(* CODESYS project CtaAppStufenManagement_1.0.0.2.library
   Description: Stufenmanagement Library der CTA
   Version: 1.0.0.2
   Title: CtaAppStufenManagement
   Author: SIS
   DocFormat: reStructuredText
   LanguageModelAttribute: qualified-access-only
   Placeholder: CtaAppStufenManagement
   DefaultNamespace: CtaAppStufenManagement
   CompiledLibraryCompatibilityVersion: CODESYS V3.5 SP16 Patch 3
   Company: CTA

Project tree, tasks and I/O mapping:
  libraries: Standard, 3.5.18.0 (System); CtaSysConfig, 1.0.0.2 (CTA); CtaSysTypes, 1.0.0.0 (CTA); CtaVisSymbols, 1.0.0.0 (CTA); CtaVisApps, 1.0.0.0 (CTA); CtaVisHelp, 1.0.0.0 (CTA); CtaVisUser, 1.0.0.0 (CTA); VisuSymbols, 4.5.0.0 (System)
  40 Visualizations/
    visualisation VIS_Manager_rEck
    Dialog/
      visualisation DIA_MANAGER
    visualisation VIS_Manager
  00000000-0000-0000-0000-000000000000|D:\CoDeSys\LibrariesV3\trunk\Intern\CAA\CAA Template\3.4.0.0 draft\Placeholder.xml
  00000000-0000-0000-0000-000000000000|D:\CoDeSys\LibrariesV3\trunk\Intern\CAA\CAA Template\3.2.0.3 draft\Prefix.pdf
  00000000-0000-0000-0000-000000000000|D:\CoDeSys\LibrariesV3\trunk\Intern\CAA\CAA Template\3.5.2.0 draft\Placeholder.xml
  20 Structs/
    data type TYPE_OF_ENGINE_MANAGEMENT
    data type scParameter
  50 Images/
  10 Documenation/
    global variables VersionHistory
    global variables readMe
  21 Interface/
    Group/
      GroupBase/
        interface ITF_GROUPBASE: IS_NOT_RELEVANT_TO_CHECK, SET_OPERATION_MODES, proiAcknowledge, prorAcknowledge, proxAcknowledge, IS_NOT_RELEVANT_TO_RELEASE, proiAvaiable, prorAvaiable, proxAvaiable, proxLockDown, IS_NOT_RELEVANT_TO_ACKNOWLEDGE
      GroupLeader/
        Circuit/
          interface ITF_CIRCUIT: GET_ANZ_AVAIABLE, GET_ANZ_ACKNOWLEDGE, GET_ANZ_RELEASE, CIRCUIT_NR, ALL_OFF, IS_RELEVANT_TO_RELEASE, GET_ENGINE_STATE, RELEASE_ENGINE, LOWERBOUND, UPPERBOUND, metSetRelease, proxRelease, GET_ANZ_LOCKDOWN, SET_HZ_SCALE, SET_ENGINE_STATE, prorRelease, proxAcknowledge
      GroupMember/
        Hydraulics/
          interface ITF_HYDRA: MEMBER_OF, IS_ADDED_TO_NESSESARY, CALCULATET_TIME_TILL_RUN, ESTIMATET_TIME_TILL_RUN, metSetRelease, proxRelease
    Manager/
      interface ITF_MANAGER: ADD_CLIENT
  11 Library Parameter/
  12 Konstanten/
    global variables GVL_CONSTANT
  60 Textlisten/
    text list TypeOfEngineManagement
  13 Globale Variablen/
  text list GlobalTextList
  5ce3da45-db07-42e7-a21c-a00fff4ed8f6|C:\Users\sis\Downloads\dip-switch.svg
  5ce3da45-db07-42e7-a21c-a00fff4ed8f6|C:\Users\sis\Downloads\lightning-bolt-circle.svg
  30 Program Organization Units/
    Group/
      GroupBase/
        function block GROUPBASE [ST]: IS_NOT_RELEVANT_TO_CHECK, SET_OPERATION_MODES, IS_NOT_RELEVANT_TO_RELEASE, proenRelease, proenCheck, proiAcknowledge, prorAcknowledge, proxAcknowledge, proiAvaiable, prorAvaiable, proxAvaiable, proxLockDown, IS_NOT_RELEVANT_TO_ACKNOWLEDGE
      GroupLeader/
        Help/
          function block ENGINE [ST]: GET_ANZ_AVAIABLE, GET_ANZ_ACKNOWLEDGE, GET_ANZ_RELEASE, GET_ANZ_LOCKDOWN, SET_ENGINE_STATE, GET_ENGINE_STATE, RELEASE_ENGINE, LOWERBOUND, UPPERBOUND, SET_HZ_SCALE
        Circuit/
          function block CIRCUIT [ST]: IS_RELEVANT_TO_RELEASE, proiAvaiable, SET_ENGINE_STATE, prorRelease, metSetRelease, proxRelease, GET_ANZ_AVAIABLE, GET_ANZ_ACKNOWLEDGE, GET_ANZ_RELEASE, CIRCUIT_NR, ALL_OFF, GET_ENGINE_STATE, RELEASE_ENGINE, LOWERBOUND, UPPERBOUND, GET_ANZ_LOCKDOWN, SET_HZ_SCALE, proxAvaiable, proxAcknowledge, proiAcknowledge
      GroupMember/
        Help/
          function block GROUPMEMBER [ST]
          function block TIME_TIL_RUN [ST]: CALCULATET_TIME_TILL_RUN, ESTIMATET_TIME_TILL_RUN
        Hydraulics/
          function block HYDRA [ST]: IS_ADDED_TO_NESSESARY, MEMBER_OF, FB_INIT, CALCULATET_TIME_TILL_RUN, ESTIMATET_TIME_TILL_RUN, metSetRelease, proxRelease
    Manager/
      function block MANAGER [ST]: GET_NEXT_ENGINE_TO_RUN, GET_NEXT_ENGINE_TO_OFF, MANAGEMENT, CHECK_RELEASE_CHANGE, UPDATE_AT_THE_END, ACKNOWLEDGE, RELEASE, LOCKDOWN, AVAIABLE, ADD_CLIENT, actParameter
  5ce3da45-db07-42e7-a21c-a00fff4ed8f6|C:\Users\sis\Downloads\sine-wave.svg
  5ce3da45-db07-42e7-a21c-a00fff4ed8f6|C:\Users\sis\Downloads\eye.svg
  5ce3da45-db07-42e7-a21c-a00fff4ed8f6|C:\Users\sis\Downloads\lan.svg
*)

// 20 Structs/TYPE_OF_ENGINE_MANAGEMENT
{attribute 'qualified_only'}
TYPE TYPE_OF_ENGINE_MANAGEMENT :
(
	RUN_1BY1 	:= 0,
	RUN_EQUAL	:= 1
);
END_TYPE

// 20 Structs/scParameter
TYPE scParameter :
	STRUCT
		fbtZuschaltSperrzeit		:	CtaSysConfig.fbTIME;
		fbiTypeOfEngineManagement	:	CtaSysConfig.fbINT;
	END_STRUCT
END_TYPE

// 10 Documenation/VersionHistory
(* 

.. image:: ../../Images/CTA_Logo.jpg
   :align: right
   :width: 15% 

**Vorlage**   


============ =========== =========== ============================================
**Date**     **Version** **Author**  **Change**
------------ ----------- ----------- --------------------------------------------
04.03.2021   0.0.0.0     SIS         Vorlage erstellt

============ =========== =========== ============================================


*)
VAR_GLOBAL
    stInfo : STRING:= '0.0.0.0, Vorlage, CTA';
END_VAR

// 10 Documenation/readMe
(*

**ReadMe**
 
|	**Empfehlung**
|
|	Die Bibliothek CtaAppStufenManagement dient dem Management der ganzen Maschine, sie Schaltet beispielsweise Kreise und Stufen frei.
|	Instanzieren Sie den CtaAppStufenManagement.MANAGER in ihrem Funktionsbaustein oder POU beispielsweise als Manager
|	Deklarieren Sie die Struktur Variable welche als Parameter und zur ansteuerung dienen wie im Code beispiel.
|  
| *Beispiel* 

+-----------------------+---------------------------------------------------------------------------------------------------------------------------------------------------------------------------------------------------------------------------------------------------------------------------------------------------------------------------------------------------------------------------------------------------------------------------------------+
| Beschreibung          |  Code                                                                                                                                                                                                                                                                                                                                                                                                                                 |
+=======================+=======================================================================================================================================================================================================================================================================================================================================================================================================================================+
| Pou oder SmFb         | .. code-block:: codesys                                                                                                                                                                                                                                                                                                                                                                                                               |
|                       |                                                                                                                                                                                                                                                                                                                                                                                                                                       |
|                       |	// Deklaration als VAR im POU oder dem selbsterstellten Funktionsbaustein                                                                                                                                                                                                                                                                                                                                                       	|
|                       |   VAR   																																																																																																								|
|						|	    (*Maschinen Management*)																																																		 																																																|
|						|		MANAGER			: CtaAppStufenManagement.MANAGER;                                                                                                                                                                                                                                                                                                                                                             				 	|
|						|																																																																																																										|
+-----------------------+---------------------------------------------------------------------------------------------------------------------------------------------------------------------------------------------------------------------------------------------------------------------------------------------------------------------------------------------------------------------------------------------------------------------------------------+
| Code für Init         | .. code-block:: codesys                                                                                                                                                                                                                                                                                                                                                                                                               |
|                       |   																																																																																																									|
| 						|	// Kopieren des nachfolgenden Codes in eine Action zur Initialisierung der Parameter. Zum Beispiel actConfig.																																																																														|
|                       |	{region "Maschinen Management"}                                                                                                                                                                                                                                                                                                                                                                                                     |
|						|		MANAGER.scParameter.fbtZuschaltSperrzeit               		(_wertInit :=	 T#5m														);		//P1 Zeit die vergeht bis die nächste Stufe zugeschalten werden kann																																																			|
|						|		MANAGER.scParameter.fbiTypeOfEngineManagement				(_wertInit :=	 	0		, _minInit :=			, _maxInit :=			);		//P2 0 = Ausschöpfung des Kreises / 1 = Beliebig nach verfügbarkeit																																																				| 
|						|	{endregion}                                                                                                                                                      																																																																	| 
+-----------------------+---------------------------------------------------------------------------------------------------------------------------------------------------------------------------------------------------------------------------------------------------------------------------------------------------------------------------------------------------------------------------------------------------------------------------------------+
*)                                                                                                                                                                                                                                                                                                                                                                                                                                                               
 VAR_GLOBAL                                                                                                                                                                                                                                                                                                                                                                                                                                                      
    xReadMeDone              :   BOOL;                                                                                                                                                                                                                                                                                                                                                                                                                           
END_VAR

// 12 Konstanten/GVL_CONSTANT
{attribute 'qualified_only'}
VAR_GLOBAL CONSTANT
	MAX_GROUPS	:	USINT	:= 4;
	MAX_ENGINE	:	USINT	:= 4;
END_VAR

// 21 Interface/Group/GroupBase/ITF_GROUPBASE
INTERFACE ITF_GROUPBASE EXTENDS __SYSTEM.IQueryInterface

PROPERTY IS_NOT_RELEVANT_TO_CHECK : BOOL
GET
END_GET
SET
END_SET
END_PROPERTY

METHOD SET_OPERATION_MODES
VAR_INPUT
	enCheckIn		:	INT;
	enReleaseIn		:	INT;
END_VAR
END_METHOD

{attribute 'monitoring' := 'call'}
PROPERTY proiAcknowledge : INT
SET
END_SET
GET
END_GET
END_PROPERTY

PROPERTY prorAcknowledge : REAL
SET
END_SET
GET
END_GET
END_PROPERTY

{attribute 'monitoring' := 'call'}
PROPERTY proxAcknowledge : BOOL
SET
END_SET
GET
END_GET
END_PROPERTY

PROPERTY IS_NOT_RELEVANT_TO_RELEASE : BOOL
GET
END_GET
SET
END_SET
END_PROPERTY

{attribute 'monitoring' := 'call'}
PROPERTY proiAvaiable : INT
SET
END_SET
GET
END_GET
END_PROPERTY

PROPERTY prorAvaiable : REAL
SET
END_SET
GET
END_GET
END_PROPERTY

{attribute 'monitoring' := 'call'}
PROPERTY proxAvaiable : BOOL
SET
END_SET
GET
END_GET
END_PROPERTY

{attribute 'monitoring' := 'call'}
PROPERTY proxLockDown : BOOL
SET
END_SET
GET
END_GET
END_PROPERTY

PROPERTY IS_NOT_RELEVANT_TO_ACKNOWLEDGE : BOOL
SET
END_SET
GET
END_GET
END_PROPERTY

END_INTERFACE

// 21 Interface/Manager/ITF_MANAGER
INTERFACE ITF_MANAGER EXTENDS __SYSTEM.IQueryInterface

METHOD ADD_CLIENT : BOOL
VAR_INPUT
	ITF_GROUP_BASE_IN	:	ITF_GROUPBASE;
END_VAR
END_METHOD

END_INTERFACE

// 21 Interface/Group/GroupLeader/Circuit/ITF_CIRCUIT
INTERFACE ITF_CIRCUIT EXTENDS ITF_GROUPBASE

PROPERTY GET_ANZ_AVAIABLE : UINT
GET
END_GET
END_PROPERTY

PROPERTY GET_ANZ_ACKNOWLEDGE : UINT
GET
END_GET
END_PROPERTY

PROPERTY GET_ANZ_RELEASE : UINT
GET
END_GET
END_PROPERTY

PROPERTY CIRCUIT_NR : USINT
GET
END_GET
END_PROPERTY

METHOD ALL_OFF : BOOL
VAR_INPUT
END_VAR
END_METHOD

PROPERTY IS_RELEVANT_TO_RELEASE : BOOL
GET
END_GET
SET
END_SET
END_PROPERTY

METHOD GET_ENGINE_STATE : BOOL
VAR_INPUT
	usiNr				:	USINT;
END_VAR
VAR_OUTPUT	    	
	xAvaiable			:	BOOL;
	xRelease			:	BOOL;
	rRelease			:	REAL;
	xAcknowledge		:	BOOL;
	rAcknowledge		:	REAL;
	xLockDown			:	BOOL;
	udiRunTime			:	UDINT;
	udiRunTimeTillOn	:	UDINT;
END_VAR
END_METHOD

METHOD RELEASE_ENGINE
VAR_INPUT
	usiNr		:	USINT;
	xRelease	:	BOOL;
END_VAR
END_METHOD

PROPERTY LOWERBOUND : DINT
GET
END_GET
END_PROPERTY

PROPERTY UPPERBOUND : DINT
GET
END_GET
END_PROPERTY

METHOD metSetRelease
VAR_INPUT
	xReleaseCircuit	:	BOOL;	
END_VAR
END_METHOD

{attribute 'monitoring' := 'call'}
PROPERTY proxRelease : BOOL
GET
END_GET
END_PROPERTY

PROPERTY GET_ANZ_LOCKDOWN : UINT
GET
END_GET
END_PROPERTY

METHOD SET_HZ_SCALE
VAR_INPUT
	scHz		:	CtaSysTypes.scHzParameter;
END_VAR
END_METHOD

METHOD SET_ENGINE_STATE 
VAR_INPUT
	usiNr		:	USINT;
	xAvaiable	:	BOOL;
	xAcknowledge:	BOOL;
	rAcknowledge:	REAL;
	xLockDown	:	BOOL;
	rNewRelease	:	REAL;
END_VAR
VAR_OUTPUT
	xRelease	:	BOOL;
	rRelease	:	REAL;
	scHz		:	CtaSysTypes.scHzParameter;
END_VAR
END_METHOD

PROPERTY prorRelease : REAL
SET
END_SET
GET
END_GET
END_PROPERTY

{attribute 'monitoring' := 'call'}
PROPERTY proxAcknowledge : BOOL
SET
END_SET
GET
END_GET
END_PROPERTY

END_INTERFACE

// 21 Interface/Group/GroupMember/Hydraulics/ITF_HYDRA
INTERFACE ITF_HYDRA EXTENDS ITF_GROUPBASE

METHOD MEMBER_OF : BOOL
VAR_INPUT
	usiGROUP_NR	:	USINT;
END_VAR
END_METHOD

PROPERTY IS_ADDED_TO_NESSESARY : BOOL
SET
END_SET
GET
END_GET
END_PROPERTY

PROPERTY CALCULATET_TIME_TILL_RUN : TIME
SET
END_SET
GET
END_GET
END_PROPERTY

PROPERTY ESTIMATET_TIME_TILL_RUN : TIME
SET
END_SET
GET
END_GET
END_PROPERTY

METHOD metSetRelease
VAR_INPUT
	usiNr		:	USINT;
	xRelease	:	BOOL;	
END_VAR
END_METHOD

{attribute 'monitoring' := 'call'}
PROPERTY proxRelease : BOOL
GET
END_GET
END_PROPERTY

END_INTERFACE

// 30 Program Organization Units/Group/GroupBase/GROUPBASE
FUNCTION_BLOCK GROUPBASE IMPLEMENTS ITF_GROUPBASE
VAR_INPUT
	ITF_MANAGER_IN			:	ITF_MANAGER;
END_VAR    
VAR_OUTPUT
	xAvaiable					:	BOOL;
	iAvaiable					:	INT;
	rAvaiable					:	REAL;
	xAcknowledge				:	BOOL;
	iAcknowledge				:	INT;
	rAcknowledge				:	REAL;
	xLockDown					:	BOOL;
END_VAR         		         		
VAR                 		
	enCheck						:	INT;
	enRelease					:	INT;	
	xIsNotRelevantToRelease		:	BOOL;
	xIsNotRelevantToCheck		:	BOOL;
	xIsNotRelevantToAcknowledge :	BOOL;
END_VAR

IF __QUERYINTERFACE(ITF_MANAGER_IN,ITF_MANAGER_IN) THEN
	ITF_MANAGER_IN.ADD_CLIENT(THIS^);	
END_IF;

PROPERTY IS_NOT_RELEVANT_TO_CHECK : BOOL
GET
IS_NOT_RELEVANT_TO_CHECK := xIsNotRelevantToCheck;
END_GET
SET
xIsNotRelevantToCheck := IS_NOT_RELEVANT_TO_CHECK;
END_SET
END_PROPERTY

METHOD SET_OPERATION_MODES
VAR_INPUT
	enCheckIn		:	INT;
	enReleaseIn		:	INT;
END_VAR
enCheck 	:= enCheckIn;
enRelease 	:= enReleaseIn;
END_METHOD

PROPERTY IS_NOT_RELEVANT_TO_RELEASE : BOOL
GET
IS_NOT_RELEVANT_TO_RELEASE := xIsNotRelevantToRelease;
END_GET
SET
xIsNotRelevantToRelease := IS_NOT_RELEVANT_TO_RELEASE;
END_SET
END_PROPERTY

{attribute 'monitoring' := 'call'}
PROPERTY proenRelease : INT
GET
proenRelease := enRelease;
END_GET
END_PROPERTY

{attribute 'monitoring' := 'call'}
PROPERTY proenCheck : INT
GET
proenCheck := enCheck;
END_GET
END_PROPERTY

{attribute 'monitoring' := 'call'}
PROPERTY proiAcknowledge : INT
SET
iAcknowledge := proiAcknowledge;
END_SET
GET
proiAcknowledge := iAcknowledge;
END_GET
END_PROPERTY

PROPERTY prorAcknowledge : REAL
SET
rAcknowledge := prorAcknowledge;
END_SET
GET
prorAcknowledge := rAcknowledge;
END_GET
END_PROPERTY

{attribute 'monitoring' := 'call'}
PROPERTY proxAcknowledge : BOOL
SET
xAcknowledge := proxAcknowledge;
END_SET
GET
proxAcknowledge := xAcknowledge;
END_GET
END_PROPERTY

{attribute 'monitoring' := 'call'}
PROPERTY proiAvaiable : INT
SET
iAvaiable := proiAvaiable;
END_SET
GET
proiAvaiable := iAvaiable;
END_GET
END_PROPERTY

PROPERTY prorAvaiable : REAL
SET
rAvaiable := prorAvaiable;
END_SET
GET
prorAvaiable := rAvaiable;
END_GET
END_PROPERTY

{attribute 'monitoring' := 'call'}
PROPERTY proxAvaiable : BOOL
SET
xAvaiable := proxAvaiable;
END_SET
GET
proxAvaiable := xAvaiable;
END_GET
END_PROPERTY

{attribute 'monitoring' := 'call'}
PROPERTY proxLockDown : BOOL
SET
xLockDown := proxLockDown;
END_SET
GET
proxLockDown := xLockDown;
END_GET
END_PROPERTY

PROPERTY IS_NOT_RELEVANT_TO_ACKNOWLEDGE : BOOL
GET
IS_NOT_RELEVANT_TO_ACKNOWLEDGE := xIsNotRelevantToAcknowledge;
END_GET
SET
xIsNotRelevantToAcknowledge := IS_NOT_RELEVANT_TO_ACKNOWLEDGE;
END_SET
END_PROPERTY

END_FUNCTION_BLOCK

// 30 Program Organization Units/Group/GroupLeader/Circuit/CIRCUIT
FUNCTION_BLOCK CIRCUIT EXTENDS GROUPBASE IMPLEMENTS ITF_CIRCUIT
VAR_INPUT
	usiNr	:	USINT;
END_VAR
VAR_OUTPUT
END_VAR
VAR
	xRelease				:	BOOL;
	rRelease				:	REAL;
	xIsRelevantToRelease	:	BOOL;
	ENGINE					:	ENGINE;
	diFor					:	DINT;
END_VAR

SUPER^();

PROPERTY IS_RELEVANT_TO_RELEASE : BOOL
SET
xIsRelevantToRelease := IS_RELEVANT_TO_RELEASE;
END_SET
GET
IS_RELEVANT_TO_RELEASE := xIsRelevantToRelease;
END_GET
END_PROPERTY

{attribute 'monitoring' := 'call'}
PROPERTY proiAvaiable : INT
SET
iAvaiable := proiAvaiable;
END_SET
GET
iAvaiable	:= TO_INT(GET_ANZ_AVAIABLE);
proiAvaiable := iAvaiable;
END_GET
END_PROPERTY

METHOD SET_ENGINE_STATE 
VAR_INPUT
	usiNr		:	USINT;
	xAvaiable	:	BOOL;
	xAcknowledge:	BOOL;
	rAcknowledge:	REAL;
	xLockDown	:	BOOL;
	rNewRelease	:	REAL;
END_VAR
VAR_OUTPUT
	xRelease	:	BOOL;
	rRelease	:	REAL;
	scHz		:	CtaSysTypes.scHzParameter;
END_VAR
ENGINE.SET_ENGINE_STATE(usiNr 			:= usiNr,
						xAvaiable 		:= xAvaiable,
						xAcknowledge	:= xAcknowledge,
						rAcknowledge	:= rAcknowledge,
						xLockDown		:= xLockDown,
						rNewRelease		:= rNewRelease,
						xRelease		=> xRelease,
						rRelease		=> rRelease,
						scHz			=> scHz);
END_METHOD

PROPERTY prorRelease : REAL
SET
rRelease := prorRelease;
END_SET
GET
prorRelease := rRelease;
END_GET
END_PROPERTY

METHOD metSetRelease
VAR_INPUT
	xReleaseCircuit	:	BOOL;	
END_VAR
xRelease := xReleaseCircuit;
IF NOT xRelease THEN
	ALL_OFF();
END_IF;
END_METHOD

{attribute 'monitoring' := 'call'}
PROPERTY proxRelease : BOOL
GET
proxRelease := xRelease;
END_GET
END_PROPERTY

PROPERTY GET_ANZ_AVAIABLE : UINT
GET
VAR
	diForTemp	:	DINT;
END_VAR
GET_ANZ_AVAIABLE := ENGINE.GET_ANZ_AVAIABLE;
END_GET
END_PROPERTY

PROPERTY GET_ANZ_ACKNOWLEDGE : UINT
GET
VAR
	diForTemp	:	DINT;
END_VAR
GET_ANZ_ACKNOWLEDGE := ENGINE.GET_ANZ_ACKNOWLEDGE;
END_GET
END_PROPERTY

PROPERTY GET_ANZ_RELEASE : UINT
GET
VAR
	diForTemp	:	DINT;
END_VAR
GET_ANZ_RELEASE := ENGINE.GET_ANZ_RELEASE;
END_GET
END_PROPERTY

PROPERTY CIRCUIT_NR : USINT
GET
CIRCUIT_NR := usiNr;
END_GET
END_PROPERTY

METHOD ALL_OFF : BOOL
VAR_INPUT
END_VAR
VAR
	diLowerBound	:	DINT;
	diUpperBound	:	DINT;
	diForTemp1		:	DINT;
END_VAR
(* Stopp ALL *)
FOR diForTemp1 := ENGINE.LOWERBOUND TO ENGINE.UPPERBOUND DO
	ENGINE.RELEASE_ENGINE(TO_USINT(diForTemp1),FALSE);
END_FOR;
END_METHOD

METHOD GET_ENGINE_STATE : BOOL
VAR_INPUT
	usiNr		:	USINT;
END_VAR
VAR_OUTPUT	    	
	xAvaiable			:	BOOL;
	xRelease			:	BOOL;
	rRelease			:	REAL;
	xAcknowledge		:	BOOL;
	rAcknowledge		:	REAL;
	xLockDown			:	BOOL;
	udiRunTime			:	UDINT;
	udiRunTimeTillOn	:	UDINT;
END_VAR
ENGINE.GET_ENGINE_STATE(usiNr 				:= usiNr,
						xAvaiable			=> xAvaiable,
						xRelease			=> xRelease,
						rRelease			=> rRelease,
						xAcknowledge		=> xAcknowledge,
						rAcknowledge		=> rAcknowledge,
						xLockDown			=> xLockDown,
						udiRunTime			=> udiRunTime,
						udiRunTimeTillOn	=> udiRunTimeTillOn);
END_METHOD

METHOD RELEASE_ENGINE
VAR_INPUT
	usiNr		:	USINT;
	xRelease	:	BOOL;
END_VAR
ENGINE.RELEASE_ENGINE(	usiNr		:= usiNr,
						xRelease 	:= xRelease);
END_METHOD

PROPERTY LOWERBOUND : DINT
GET
LOWERBOUND := ENGINE.LOWERBOUND;
END_GET
END_PROPERTY

PROPERTY UPPERBOUND : DINT
GET
UPPERBOUND := ENGINE.UPPERBOUND;
END_GET
END_PROPERTY

PROPERTY GET_ANZ_LOCKDOWN : UINT
GET
GET_ANZ_LOCKDOWN := ENGINE.GET_ANZ_LOCKDOWN;
END_GET
END_PROPERTY

METHOD SET_HZ_SCALE
VAR_INPUT
	scHz		:	CtaSysTypes.scHzParameter;
END_VAR
ENGINE.SET_HZ_SCALE(scHz);
END_METHOD

{attribute 'monitoring' := 'call'}
PROPERTY proxAvaiable : BOOL
SET
xAvaiable := proxAvaiable;
END_SET
GET
proxAvaiable := SUPER^.proxAvaiable;
END_GET
END_PROPERTY

{attribute 'monitoring' := 'call'}
PROPERTY proxAcknowledge : BOOL
SET
xAcknowledge := proxAcknowledge;
END_SET
GET
proxAcknowledge := xAcknowledge;
END_GET
END_PROPERTY

{attribute 'monitoring' := 'call'}
PROPERTY proiAcknowledge : INT
SET
iAcknowledge := proiAcknowledge;
END_SET
GET
iAcknowledge := TO_INT(GET_ANZ_ACKNOWLEDGE);
proiAcknowledge := iAcknowledge;
END_GET
END_PROPERTY

END_FUNCTION_BLOCK

// 30 Program Organization Units/Group/GroupLeader/Help/ENGINE
FUNCTION_BLOCK ENGINE
VAR_INPUT
END_VAR
VAR_OUTPUT
END_VAR
VAR
	scHzAll				:	CtaSysTypes.scHzParameter;
	AY_XRELEASE			:	ARRAY[1..GVL_CONSTANT.MAX_ENGINE] OF BOOL;
	AY_RRELEASE			:	ARRAY[1..GVL_CONSTANT.MAX_ENGINE] OF REAL;
	AY_XAVAIABLE		:	ARRAY[1..GVL_CONSTANT.MAX_ENGINE] OF BOOL;
	AY_XACKNOWLEDGE		:	ARRAY[1..GVL_CONSTANT.MAX_ENGINE] OF BOOL;
	AY_XACKNOWLEDGEOLD	:	ARRAY[1..GVL_CONSTANT.MAX_ENGINE] OF BOOL;
	AY_RACKNOWLEDGE		:	ARRAY[1..GVL_CONSTANT.MAX_ENGINE] OF REAL;
	AY_LOCKDOWN			:	ARRAY[1..GVL_CONSTANT.MAX_ENGINE] OF BOOL;
	AY_RUN_TIME			:	ARRAY[1..GVL_CONSTANT.MAX_ENGINE] OF UDINT;
	AY_RUN_TIME_TILL_ON	:	ARRAY[1..GVL_CONSTANT.MAX_ENGINE] OF UDINT;
	AY_TON_RUN_TIME		:	ARRAY[1..GVL_CONSTANT.MAX_ENGINE] OF Standard.TON;
END_VAR

PROPERTY GET_ANZ_AVAIABLE : UINT
GET
VAR
	diForTemp	:	DINT;
END_VAR
GET_ANZ_AVAIABLE := 0;
FOR diForTemp := LOWER_BOUND(AY_XAVAIABLE,1) TO UPPER_BOUND(AY_XAVAIABLE,1) DO
	IF AY_XAVAIABLE[diForTemp] THEN
		GET_ANZ_AVAIABLE := GET_ANZ_AVAIABLE + 1;
	END_IF;
END_FOR;
END_GET
END_PROPERTY

PROPERTY GET_ANZ_ACKNOWLEDGE : UINT
GET
VAR
	diForTemp	:	DINT;
END_VAR
GET_ANZ_ACKNOWLEDGE := 0;
FOR diForTemp := LOWER_BOUND(AY_XACKNOWLEDGE,1) TO UPPER_BOUND(AY_XACKNOWLEDGE,1) DO
	IF AY_XACKNOWLEDGE[diForTemp] THEN
		GET_ANZ_ACKNOWLEDGE := GET_ANZ_ACKNOWLEDGE + 1;
	END_IF;
END_FOR;
END_GET
END_PROPERTY

PROPERTY GET_ANZ_RELEASE : UINT
GET
VAR
	diForTemp	:	DINT;
END_VAR
GET_ANZ_RELEASE := 0;
FOR diForTemp := LOWER_BOUND(AY_XRELEASE,1) TO UPPER_BOUND(AY_XRELEASE,1) DO
	IF AY_XRELEASE[diForTemp] THEN
		GET_ANZ_RELEASE := GET_ANZ_RELEASE + 1;
	END_IF;
END_FOR;
END_GET
END_PROPERTY

PROPERTY GET_ANZ_LOCKDOWN : UINT
GET
VAR
	diForTemp	:	DINT;
END_VAR
GET_ANZ_LOCKDOWN := 0;
FOR diForTemp := LOWER_BOUND(AY_LOCKDOWN,1) TO UPPER_BOUND(AY_LOCKDOWN,1) DO
	IF AY_LOCKDOWN[diForTemp] THEN
		GET_ANZ_LOCKDOWN := GET_ANZ_LOCKDOWN + 1;
	END_IF;
END_FOR;
END_GET
END_PROPERTY

METHOD SET_ENGINE_STATE 
VAR_INPUT
	usiNr		:	USINT;
	xAvaiable	:	BOOL;
	xAcknowledge:	BOOL;
	rAcknowledge:	REAL;
	xLockDown	:	BOOL;
	rNewRelease	:	REAL;
END_VAR
VAR_OUTPUT
	xRelease	:	BOOL;
	rRelease	:	REAL;
	scHz		:	CtaSysTypes.scHzParameter;
END_VAR
(* Avaiable *)
IF usiNr >= LOWER_BOUND(AY_XAVAIABLE,1) AND usiNr <= UPPER_BOUND(AY_XAVAIABLE,1) THEN
	AY_XAVAIABLE[usiNr] := xAvaiable;
END_IF;

(* Acknowledge *)
IF usiNr >= LOWER_BOUND(AY_XACKNOWLEDGE,1) AND usiNr <= UPPER_BOUND(AY_XACKNOWLEDGE,1) THEN
	AY_XACKNOWLEDGEOLD[usiNr] 	:= AY_XACKNOWLEDGE[usiNr];
	AY_XACKNOWLEDGE[usiNr] 		:= xAcknowledge;
END_IF;
IF usiNr >= LOWER_BOUND(AY_RACKNOWLEDGE,1) AND usiNr <= UPPER_BOUND(AY_RACKNOWLEDGE,1) THEN
	AY_RACKNOWLEDGE[usiNr] := rAcknowledge;
END_IF

(* LockDown *)
IF usiNr >= LOWER_BOUND(AY_LOCKDOWN,1) AND usiNr <= UPPER_BOUND(AY_LOCKDOWN,1) THEN
	AY_LOCKDOWN[usiNr] := xLockDown;
	IF xLockDown THEN
		AY_XRELEASE[usiNr] := FALSE;
	END_IF;
END_IF;

(* Release *)
IF usiNr >= LOWER_BOUND(AY_XRELEASE,1) AND usiNr <= UPPER_BOUND(AY_XRELEASE,1) THEN
	(* No release if no more acknowledge *)
	IF AY_XRELEASE[usiNr] AND AY_XRELEASE[usiNr] = AY_XACKNOWLEDGEOLD[usiNr] AND NOT AY_XACKNOWLEDGE[usiNr] THEN
		AY_XRELEASE[usiNr] := FALSE;
	END_IF;	
	xRelease := AY_XRELEASE[usiNr] AND NOT xLockDown;
ELSE
	xRelease := FALSE;
END_IF;
IF usiNr >= LOWER_BOUND(AY_RRELEASE,1) AND usiNr <= UPPER_BOUND(AY_RRELEASE,1) THEN
	AY_RRELEASE[usiNr]	:= rNewRelease;
	rRelease 			:= AY_RRELEASE[usiNr];
ELSE
	rRelease := 0;
END_IF;

(* TIME *)
IF usiNr >= LOWER_BOUND(AY_RUN_TIME,1) AND usiNr <= UPPER_BOUND(AY_RUN_TIME,1) THEN
	AY_TON_RUN_TIME[usiNr](IN := NOT AY_TON_RUN_TIME[usiNr].Q AND xRelease AND xAcknowledge,
						   PT := T#1M);
	IF AY_TON_RUN_TIME[usiNr].Q THEN
		AY_RUN_TIME[usiNr] 			:= AY_RUN_TIME[usiNr] + 1;
		AY_RUN_TIME_TILL_ON[usiNr] 	:= AY_RUN_TIME_TILL_ON[usiNr] + 1;
	END_IF;
	IF NOT xRelease THEN
		AY_RUN_TIME_TILL_ON[usiNr] 	:= 0;
	END_IF;
END_IF;

scHz := scHzAll;
END_METHOD

METHOD GET_ENGINE_STATE : BOOL
VAR_INPUT
	usiNr			:	USINT;
END_VAR         	
VAR_OUTPUT	    	
	xAvaiable			:	BOOL;
	xRelease			:	BOOL;
	rRelease			:	REAL;
	xAcknowledge		:	BOOL;
	rAcknowledge		:	REAL;
	xLockDown			:	BOOL;
	udiRunTime			:	UDINT;
	udiRunTimeTillOn	:	UDINT;
END_VAR
(* Avaiable *)
IF usiNr >= LOWER_BOUND(AY_XAVAIABLE,1) AND usiNr <= UPPER_BOUND(AY_XAVAIABLE,1) THEN
	xAvaiable := AY_XAVAIABLE[usiNr];
END_IF;

(* Release *)
IF usiNr >= LOWER_BOUND(AY_XRELEASE,1) AND usiNr <= UPPER_BOUND(AY_XRELEASE,1) THEN
	xRelease := AY_XRELEASE[usiNr];
END_IF;

(* Release *)
IF usiNr >= LOWER_BOUND(AY_RRELEASE,1) AND usiNr <= UPPER_BOUND(AY_RRELEASE,1) THEN
	rRelease := AY_RRELEASE[usiNr];
END_IF;

(* Acknowledge *)
IF usiNr >= LOWER_BOUND(AY_XACKNOWLEDGE,1) AND usiNr <= UPPER_BOUND(AY_XACKNOWLEDGE,1) THEN
	xAcknowledge := AY_XACKNOWLEDGE[usiNr];
END_IF;
IF usiNr >= LOWER_BOUND(AY_RACKNOWLEDGE,1) AND usiNr <= UPPER_BOUND(AY_RACKNOWLEDGE,1) THEN
	rAcknowledge := AY_RACKNOWLEDGE[usiNr];
END_IF

(* LockDown *)
IF usiNr >= LOWER_BOUND(AY_LOCKDOWN,1) AND usiNr <= UPPER_BOUND(AY_LOCKDOWN,1) THEN
	xLockDown := AY_LOCKDOWN[usiNr];
END_IF;

(* Temp Min Run *)
IF usiNr >= LOWER_BOUND(AY_RUN_TIME,1) AND usiNr <= UPPER_BOUND(AY_RUN_TIME,1) THEN
	udiRunTime := AY_RUN_TIME[usiNr];
END_IF;

(* Temp Min Run Till On*)
IF usiNr >= LOWER_BOUND(AY_RUN_TIME_TILL_ON,1) AND usiNr <= UPPER_BOUND(AY_RUN_TIME_TILL_ON,1) THEN
	udiRunTimeTillOn := AY_RUN_TIME_TILL_ON[usiNr];
END_IF;
END_METHOD

METHOD RELEASE_ENGINE : BOOL
VAR_INPUT
	usiNr		:	USINT;
	xRelease	:	BOOL;
END_VAR
(* Release *)
IF usiNr >= LOWER_BOUND(AY_XRELEASE,1) AND usiNr <= UPPER_BOUND(AY_XRELEASE,1) THEN
	AY_XRELEASE[usiNr] := xRelease;
	IF NOT xRelease THEN
		AY_RRELEASE[usiNr] := 0;
	END_IF;
END_IF;
END_METHOD

PROPERTY LOWERBOUND : DINT
GET
LOWERBOUND := LOWER_BOUND(AY_XRELEASE,1);
END_GET
END_PROPERTY

PROPERTY UPPERBOUND : DINT
GET
UPPERBOUND := UPPER_BOUND(AY_XRELEASE,1);
END_GET
END_PROPERTY

METHOD SET_HZ_SCALE
VAR_INPUT
	scHz		:	CtaSysTypes.scHzParameter;
END_VAR
scHzAll := scHz;
END_METHOD

END_FUNCTION_BLOCK

// 30 Program Organization Units/Group/GroupMember/Help/GROUPMEMBER
FUNCTION_BLOCK GROUPMEMBER
VAR_INPUT
	AY_MEMBER_OF		:	ARRAY[0..4] OF BOOL;
END_VAR
VAR_OUTPUT
	xTrigIsChanged		:	BOOL;
END_VAR
VAR
	AY_MEMBER_OF_OLD	:	ARRAY[0..4] OF BOOL;
	diFor1				:	DINT;
END_VAR

xTrigIsChanged := FALSE;
FOR diFor1 := LOWER_BOUND(AY_MEMBER_OF,1) TO UPPER_BOUND(AY_MEMBER_OF,1) DO
	IF AY_MEMBER_OF[diFor1] <> AY_MEMBER_OF_OLD[diFor1] THEN
		xTrigIsChanged 				:= TRUE;
		AY_MEMBER_OF_OLD[diFor1]	:= AY_MEMBER_OF[diFor1];
	END_IF
END_FOR;

END_FUNCTION_BLOCK

// 30 Program Organization Units/Group/GroupMember/Help/TIME_TIL_RUN
FUNCTION_BLOCK TIME_TIL_RUN
VAR_INPUT
END_VAR
VAR_OUTPUT
END_VAR
VAR
	T_CT_TILL_RUN	:	TIME;	(* Calculatet Time till Run *)
	T_ET_TILL_RUN	:	TIME;	(* Estimatet Time till Run *)	
END_VAR

PROPERTY CALCULATET_TIME_TILL_RUN : TIME
SET
T_CT_TILL_RUN := CALCULATET_TIME_TILL_RUN;
END_SET
GET
CALCULATET_TIME_TILL_RUN := T_CT_TILL_RUN;
END_GET
END_PROPERTY

PROPERTY ESTIMATET_TIME_TILL_RUN : TIME
SET
T_ET_TILL_RUN := ESTIMATET_TIME_TILL_RUN;
END_SET
GET
ESTIMATET_TIME_TILL_RUN := T_ET_TILL_RUN;
END_GET
END_PROPERTY

END_FUNCTION_BLOCK

// 30 Program Organization Units/Group/GroupMember/Hydraulics/HYDRA
FUNCTION_BLOCK HYDRA EXTENDS GROUPBASE IMPLEMENTS ITF_HYDRA
VAR_OUTPUT
END_VAR
VAR
	xIsAddedToNessesary	:	BOOL;
	ayxRelease			:	ARRAY[1..GVL_CONSTANT.MAX_GROUPS] OF BOOL;
	GROUPMEMBER			:	GROUPMEMBER;
	TIME_TIL_RUN		:	TIME_TIL_RUN;
END_VAR

SUPER^();
GROUPMEMBER();
IF GROUPMEMBER.xTrigIsChanged THEN
	xIsAddedToNessesary := FALSE;
END_IF;

PROPERTY IS_ADDED_TO_NESSESARY : BOOL
GET
IS_ADDED_TO_NESSESARY := xIsAddedToNessesary;
END_GET
SET
xIsAddedToNessesary := IS_ADDED_TO_NESSESARY;
END_SET
END_PROPERTY

METHOD MEMBER_OF : BOOL
VAR_INPUT
	usiGROUP_NR	: USINT;
END_VAR
IF usiGROUP_NR >= LOWER_BOUND(GROUPMEMBER.AY_MEMBER_OF,1) AND usiGROUP_NR <= UPPER_BOUND(GROUPMEMBER.AY_MEMBER_OF,1) THEN
	IF GROUPMEMBER.AY_MEMBER_OF[0] THEN
		MEMBER_OF := TRUE;
	ELSE
		MEMBER_OF := GROUPMEMBER.AY_MEMBER_OF[usiGROUP_NR];
	END_IF
ELSE
	MEMBER_OF := FALSE;
END_IF;
END_METHOD

//FB_Init ist immer implizit verfügbar und wird primär für die Initialisierung verwendet.
//Der Rückgabewert wird nicht ausgewertet. Für gezielte Einflussnahme können Sie
//die Methoden explizit deklarieren und darin mit dem Standard-Initialisierungscode 
//zusätzlichen Code bereitstellen. Sie können den Rückgabewert auswerten.
METHOD FB_Init: BOOL
VAR_INPUT    
bInitRetains: BOOL; // TRUE: Die Retain-Variablen werden initialisiert (Reset warm / Reset kalt)    
bInCopyCode: BOOL;  // TRUE: Die Instanz wird danach in den Kopiercode kopiert (Online-Change)
END_VAR
VAR_INPUT
	xAll	:	BOOL;
	xGp1	:	BOOL;
	xGp2	:	BOOL;
	xGp3	:	BOOL;
	xGp4	:	BOOL;
END_VAR
GROUPMEMBER.AY_MEMBER_OF[0] := xAll;
GROUPMEMBER.AY_MEMBER_OF[1] := xGp1;
GROUPMEMBER.AY_MEMBER_OF[2] := xGp2;
GROUPMEMBER.AY_MEMBER_OF[3]	:= xGp3;
GROUPMEMBER.AY_MEMBER_OF[4]	:= xGp4;
END_METHOD

PROPERTY CALCULATET_TIME_TILL_RUN : TIME
SET
TIME_TIL_RUN.CALCULATET_TIME_TILL_RUN := CALCULATET_TIME_TILL_RUN;
END_SET
GET
CALCULATET_TIME_TILL_RUN := TIME_TIL_RUN.CALCULATET_TIME_TILL_RUN;
END_GET
END_PROPERTY

PROPERTY ESTIMATET_TIME_TILL_RUN : TIME
SET
TIME_TIL_RUN.ESTIMATET_TIME_TILL_RUN := ESTIMATET_TIME_TILL_RUN;
END_SET
GET
ESTIMATET_TIME_TILL_RUN := TIME_TIL_RUN.ESTIMATET_TIME_TILL_RUN;
END_GET
END_PROPERTY

METHOD metSetRelease
VAR_INPUT
	usiNr		:	USINT;
	xRelease	:	BOOL;	
END_VAR
IF usiNr >= LOWER_BOUND(ayxRelease,1) AND usiNr <= UPPER_BOUND(ayxRelease,1) THEN
	ayxRelease[usiNr] := xRelease;
END_IF;
END_METHOD

{attribute 'monitoring' := 'call'}
PROPERTY proxRelease : BOOL
GET
VAR
	diForTemp	:	DINT;
END_VAR
proxRelease :=  FALSE; 
FOR diForTemp := LOWER_BOUND(ayxRelease,1) TO UPPER_BOUND(ayxRelease,1) DO
	IF ayxRelease[diForTemp] THEN
		proxRelease :=  TRUE;
	END_IF;	
END_FOR;
END_GET
END_PROPERTY

END_FUNCTION_BLOCK

// 30 Program Organization Units/Manager/MANAGER
FUNCTION_BLOCK MANAGER IMPLEMENTS ITF_MANAGER
VAR_INPUT
	enCheck							:	INT;
	xRelease						:	BOOL;
	iRelease						:	INT;
	rRelease						:	REAL;
	enRelease						:	INT;
	scHzRelease						:	CtaSysTypes.scHzParameter;
END_VAR         					
VAR_OUTPUT      					
	xAvaiable						:	BOOL;
	iAvaiable						:	INT;
	xAcknowledge					: 	BOOL;
	iAcknowledge					:	INT;
	rAcknowledge					:	REAL;
	xLockDown						:	BOOL;
	ITF_MANAGER						:	ITF_MANAGER;
END_VAR         					
VAR     					
	aydiSyncG						:	ARRAY[1..GVL_CONSTANT.MAX_GROUPS] OF DINT :=[GVL_CONSTANT.MAX_GROUPS(1)];
	AY_GROUPS						:	ARRAY[1..GVL_CONSTANT.MAX_GROUPS] OF ARRAY[0..20] OF ITF_GROUPBASE;
	AY_GROUPS_xAVAIABLE				:	ARRAY[1..GVL_CONSTANT.MAX_GROUPS] OF BOOL;
	AY_GROUPS_iAVAIABLE				:	ARRAY[1..GVL_CONSTANT.MAX_GROUPS] OF INT;
	AY_GROUPS_xACKNOWLEDG			:	ARRAY[1..GVL_CONSTANT.MAX_GROUPS] OF BOOL;
	AY_GROUPS_iACKNOWLEDG			:	ARRAY[1..GVL_CONSTANT.MAX_GROUPS] OF INT;
	AY_GROUPS_rACKNOWLEDG			:	ARRAY[1..GVL_CONSTANT.MAX_GROUPS] OF REAL;
	AY_GROUPS_xLOCKDOWN				:	ARRAY[1..GVL_CONSTANT.MAX_GROUPS] OF BOOL;
	AY_GROUPS_xRELEASE				:	ARRAY[1..GVL_CONSTANT.MAX_GROUPS] OF BOOL;
	AY_GROUPS_iRELEASE				:	ARRAY[1..GVL_CONSTANT.MAX_GROUPS] OF INT;
	AY_GROUPS_rRELEASE				:	ARRAY[1..GVL_CONSTANT.MAX_GROUPS] OF REAL;
	AY_GROUPS_AyPosMaxCT			:	ARRAY[1..GVL_CONSTANT.MAX_GROUPS] OF DINT;
	AY_GROUPS_xReleaseCircuit		:	ARRAY[1..GVL_CONSTANT.MAX_GROUPS] OF BOOL;
	T_Temp_Max_CT					:	TIME;
	TEMP_ITF_CIRCUIT				:	ITF_CIRCUIT;
	TEMP_ITF_HYDRA					:	ITF_HYDRA;
	TEMP_ITF_HYDRA_MAX_CT			:	ITF_HYDRA;
	diTempMemberCount				:	DINT;
	diFor1							:	DINT;
	diFor2							:	DINT;
	diNextCircuitToRun  			: 	DINT;
	diNextEngineToRun				: 	DINT;		
	diNextCircuitToOff  			: 	DINT;
	diNextEngineToOff				: 	DINT;	
	xTrigOn							:	BOOL;
	xTrigOff						: 	BOOL;
	iTrigOffCount					:	INT;
	iTrigOffMax						:	INT;
	enCheckOld						:	INT;
	enReleaseOld					:	INT;
	uiCountGroupLockDown			:	UINT;
	uiCountEngineLockDown			:	UINT;
	uiCountEngineAcknowledge		:	UINT;
	uiCountGroupLockDownOld			:	UINT;
	uiCountEngineAcknowledgeOld		:	UINT;
	uiCountEngineLockDownOld		:	UINT;
	iReleaseOld						:	INT;
	iAcknowledgeOld					:	INT;
	xReleaseStopp					:	BOOL;
	TP_ReleaseLock					:	Standard.TP;
	xResettReleaseLock_VIS			:	BOOL;
	// Parameter
	fbConfigFile 					:	CtaSysConfig.fbConfigFile;
	scParameter						:	scParameter;
END_VAR

actParameter();

(* ITF *)
ITF_MANAGER := THIS^;

(* AVAIABLE *)
AVAIABLE(); 

(* LOCKDOWN *)
LOCKDOWN();

(* ACKNOWLEDGE *)
ACKNOWLEDGE();

(* MANAGEMENT *)
MANAGEMENT();

(* RELEASE *)
RELEASE();

(* CHECK CHANGE *)
CHECK_RELEASE_CHANGE();

(* UPDATE *)
UPDATE_AT_THE_END();

METHOD GET_NEXT_ENGINE_TO_RUN 
VAR_INPUT
	enTYPE_OF_ENGINE_MANAGEMENT	:	TYPE_OF_ENGINE_MANAGEMENT;
END_VAR
VAR_OUTPUT
	diNextCircuitToRunOut  		: DINT;
	diNextEngineToRunOut		: DINT;	
END_VAR
VAR 
	_diNextCircuitToRun  		: DINT;
	_diEngineLowestRunTime		: DINT;
	_xAvaiable					: BOOL;
	_xRelease					: BOOL;
	_rRelease					: REAL;
	_xAcknowledge				: BOOL;
	_rAcknowledge				: REAL;
	_xLockDown					: BOOL;
	_udiRunTime		    		: UDINT;
	_udiRunTimeTillOn   		: UDINT;
	_udiMinRunTime				: UDINT;
	_uiLowestWorkloadCircuit	: UINT;
END_VAR
(* Set Min Run Time To Max *)
_udiMinRunTime := 16#FFFFFFFF;
(* Set Lowest Workload Circuit to MAX *)
_uiLowestWorkloadCircuit := 16#FFFF;
(* Set Circuit to 0 *)
_diNextCircuitToRun := 0;
diNextCircuitToRunOut := 0;
(* Set Engine to 0  *)
_diEngineLowestRunTime := 0;
diNextEngineToRunOut := 0;

IF enTYPE_OF_ENGINE_MANAGEMENT = TYPE_OF_ENGINE_MANAGEMENT.RUN_1BY1 THEN
	FOR diFor1 := UPPER_BOUND(AY_GROUPS,1) TO LOWER_BOUND(AY_GROUPS,1) BY -1 DO 
		(* If No Error avaiable to release*)
		IF NOT AY_GROUPS_xLOCKDOWN[diFor1] AND (AY_GROUPS_xAVAIABLE[diFor1] OR AY_GROUPS_xACKNOWLEDG[diFor1]) THEN	
			IF __QUERYINTERFACE(AY_GROUPS[diFor1][LOWER_BOUND(AY_GROUPS[diFor1],1)],TEMP_ITF_CIRCUIT) THEN
				IF TEMP_ITF_CIRCUIT.GET_ANZ_RELEASE > 0 AND TEMP_ITF_CIRCUIT.GET_ANZ_AVAIABLE > 0 THEN
					(* iterate Engine and Check if Avaiable and get the Minits *)
					FOR diFor2 := TEMP_ITF_CIRCUIT.UPPERBOUND TO TEMP_ITF_CIRCUIT.LOWERBOUND BY -1 DO
						TEMP_ITF_CIRCUIT.GET_ENGINE_STATE(	usiNr 			:= TO_USINT(diFor2),
															xAvaiable 		=> _xAvaiable,
															xRelease		=> _xRelease,
															rRelease		=> _rRelease,
															xAcknowledge 	=> _xAcknowledge,
															rAcknowledge 	=> _rAcknowledge,
															xLockDown 		=> _xLockDown,
															udiRunTime 		=> _udiRunTime,
															udiRunTimeTillOn=> _udiRunTimeTillOn);
						(* Get time if Avaiable *)
						IF _xAvaiable AND NOT _xRelease AND NOT _xLockDown THEN
							IF _udiRunTime <= _udiMinRunTime THEN
								_udiMinRunTime 			:= _udiRunTime;
								_diNextCircuitToRun 	:= diFor1;
								_diEngineLowestRunTime  := diFor2;
							END_IF;			
						END_IF;						
					END_FOR;
				END_IF;
			END_IF;
		END_IF;
	END_FOR;
	(* Get new Ccuit if not possible to add ad running circuti *)
	IF _diNextCircuitToRun = 0 AND _diEngineLowestRunTime = 0  THEN
		FOR diFor1 := UPPER_BOUND(AY_GROUPS,1) TO LOWER_BOUND(AY_GROUPS,1) BY -1 DO
			(* If No Error avaiable to release*)
			IF NOT AY_GROUPS_xLOCKDOWN[diFor1] AND (AY_GROUPS_xAVAIABLE[diFor1] OR AY_GROUPS_xACKNOWLEDG[diFor1]) THEN	
				IF __QUERYINTERFACE(AY_GROUPS[diFor1][LOWER_BOUND(AY_GROUPS[diFor1],1)],TEMP_ITF_CIRCUIT) THEN
					IF TEMP_ITF_CIRCUIT.GET_ANZ_AVAIABLE > 0 THEN
						(* iterate Engine and Check if Avaiable and get the Minits *)
						FOR diFor2 := TEMP_ITF_CIRCUIT.UPPERBOUND TO TEMP_ITF_CIRCUIT.LOWERBOUND BY -1 DO
							TEMP_ITF_CIRCUIT.GET_ENGINE_STATE(	usiNr 			:= TO_USINT(diFor2),
																xAvaiable 		=> _xAvaiable,
																xRelease		=> _xRelease,
																rRelease		=> _rRelease,
																xAcknowledge 	=> _xAcknowledge,
																rAcknowledge 	=> _rAcknowledge,
																xLockDown 		=> _xLockDown,
																udiRunTime 		=> _udiRunTime,
																udiRunTimeTillOn=> _udiRunTimeTillOn);
							(* Get time if Avaiable *)
							IF _xAvaiable AND NOT _xRelease AND NOT _xLockDown THEN
								IF _udiRunTime <= _udiMinRunTime THEN
									_udiMinRunTime 			:= _udiRunTime;
									_diNextCircuitToRun 	:= diFor1;
									_diEngineLowestRunTime  := diFor2;
								END_IF;			
							END_IF;						
						END_FOR;
					END_IF;
				END_IF;
			END_IF;
		END_FOR;		
	END_IF
(* EQUAL *)
ELSIF enTYPE_OF_ENGINE_MANAGEMENT = TYPE_OF_ENGINE_MANAGEMENT.RUN_EQUAL THEN
	FOR diFor1 := UPPER_BOUND(AY_GROUPS,1) TO LOWER_BOUND(AY_GROUPS,1) BY -1 DO 
		(* If No Error avaiable to release*)
		IF NOT AY_GROUPS_xLOCKDOWN[diFor1] AND (AY_GROUPS_xAVAIABLE[diFor1] OR AY_GROUPS_xACKNOWLEDG[diFor1]) THEN	
			IF __QUERYINTERFACE(AY_GROUPS[diFor1][LOWER_BOUND(AY_GROUPS[diFor1],1)],TEMP_ITF_CIRCUIT) THEN
				IF TEMP_ITF_CIRCUIT.GET_ANZ_RELEASE <= _uiLowestWorkloadCircuit AND TEMP_ITF_CIRCUIT.GET_ANZ_AVAIABLE > 0 THEN
					_uiLowestWorkloadCircuit := TEMP_ITF_CIRCUIT.GET_ANZ_RELEASE; 
					(* iterate Engine and Check if Avaiable and get the Minits *)
					FOR diFor2 := TEMP_ITF_CIRCUIT.UPPERBOUND TO TEMP_ITF_CIRCUIT.LOWERBOUND BY -1 DO
						TEMP_ITF_CIRCUIT.GET_ENGINE_STATE(	usiNr 			:= TO_USINT(diFor2),
															xAvaiable 		=> _xAvaiable,
															xRelease		=> _xRelease,
															rRelease		=> _rRelease,
															xAcknowledge 	=> _xAcknowledge,
															rAcknowledge 	=> _rAcknowledge,
															xLockDown 		=> _xLockDown,
															udiRunTime 		=> _udiRunTime,
															udiRunTimeTillOn=> _udiRunTimeTillOn);
						(* Get time if Avaiable *)
						IF _xAvaiable AND NOT _xRelease AND NOT _xLockDown THEN
							IF _udiRunTime <= _udiMinRunTime THEN
								_udiMinRunTime 			:= _udiRunTime;
								_diNextCircuitToRun 	:= diFor1;
								_diEngineLowestRunTime  := diFor2;
							END_IF;			
						END_IF;						
					END_FOR;
				END_IF;
			END_IF;
		END_IF;
	END_FOR;
END_IF;
diNextCircuitToRunOut 	:= _diNextCircuitToRun;
diNextEngineToRunOut	:= _diEngineLowestRunTime;
END_METHOD

METHOD GET_NEXT_ENGINE_TO_OFF 
VAR_INPUT
	enTYPE_OF_ENGINE_MANAGEMENT	:	TYPE_OF_ENGINE_MANAGEMENT;
END_VAR
VAR_OUTPUT
	diNextCircuitToOffOut  		: DINT;
	diNextEngineToOffOut		: DINT;	
END_VAR
VAR 
	_diNextCircuitToOff  		: DINT;
	_diEngineHighestRunTime		: DINT;
	_xAvaiable					: BOOL;
	_xRelease					: BOOL;
	_rRelease					: REAL;
	_xAcknowledge				: BOOL;
	_rAcknowledge				: REAL;
	_xLockDown					: BOOL;
	_udiRunTime		    		: UDINT;
	_udiRunTimeTillOn   		: UDINT;
	_udiMaxRunTimeTillOn		: UDINT;
	_uiHighestWorkloadCircuit	: UINT;
	_uiLowestWorkloadCircuit	: UINT;
END_VAR
(* Set Lowest Workload Circuit to Min *)
_uiHighestWorkloadCircuit := 16#0000;
(* Set Lowest Workload Circuit to MAX *)
_uiLowestWorkloadCircuit := 16#FFFF;
(* Set Max Run Time To Min *)
_udiMaxRunTimeTillOn := 16#0000;
(* Set Circuit to 0 *)
_diNextCircuitToOff := 0;
diNextCircuitToOffOut := 0;
(* Set Engine to 0  *)
_diEngineHighestRunTime := 0;
diNextEngineToOffOut := 0;
(* 1By1 *)
IF enTYPE_OF_ENGINE_MANAGEMENT = TYPE_OF_ENGINE_MANAGEMENT.RUN_1BY1 THEN
	FOR diFor1 := UPPER_BOUND(AY_GROUPS,1) TO LOWER_BOUND(AY_GROUPS,1) BY -1 DO 
		(* If No Error avaiable to release*)
		IF NOT AY_GROUPS_xLOCKDOWN[diFor1] THEN	
			IF __QUERYINTERFACE(AY_GROUPS[diFor1][LOWER_BOUND(AY_GROUPS[diFor1],1)],TEMP_ITF_CIRCUIT) THEN
				IF TEMP_ITF_CIRCUIT.GET_ANZ_RELEASE > 0 THEN
					IF TEMP_ITF_CIRCUIT.GET_ANZ_RELEASE <= _uiLowestWorkloadCircuit THEN
						IF TEMP_ITF_CIRCUIT.GET_ANZ_RELEASE < _uiLowestWorkloadCircuit THEN
							_uiLowestWorkloadCircuit := TEMP_ITF_CIRCUIT.GET_ANZ_RELEASE; 
							(* Set Max Run Time To Min *)
							_udiMaxRunTimeTillOn := 16#0000;
						END_IF;

						(* iterate Engine and Check if Avaiable and get the Minits *)
						FOR diFor2 := TEMP_ITF_CIRCUIT.UPPERBOUND TO TEMP_ITF_CIRCUIT.LOWERBOUND BY -1 DO
							TEMP_ITF_CIRCUIT.GET_ENGINE_STATE(	usiNr 			:= TO_USINT(diFor2),
																xAvaiable 		=> _xAvaiable,
																xRelease		=> _xRelease,
																rRelease		=> _rRelease,
																xAcknowledge 	=> _xAcknowledge,
																rAcknowledge 	=> _rAcknowledge,
																xLockDown 		=> _xLockDown,
																udiRunTime 		=> _udiRunTime,
																udiRunTimeTillOn=> _udiRunTimeTillOn);
							(* Get time if Running *)
							IF _xRelease THEN
								IF _udiRunTimeTillOn >= _udiMaxRunTimeTillOn THEN
									_udiMaxRunTimeTillOn 	:= _udiRunTimeTillOn;
									_diNextCircuitToOff 	:= diFor1;
									_diEngineHighestRunTime := diFor2;
								END_IF;			
							END_IF;						
						END_FOR;
					END_IF;
				END_IF;
			END_IF;
		END_IF;
	END_FOR;
(* EQUAL *)
ELSIF enTYPE_OF_ENGINE_MANAGEMENT = TYPE_OF_ENGINE_MANAGEMENT.RUN_EQUAL THEN
	FOR diFor1 := UPPER_BOUND(AY_GROUPS,1) TO LOWER_BOUND(AY_GROUPS,1) BY -1 DO 
		(* If No Error avaiable to release*)
		IF NOT AY_GROUPS_xLOCKDOWN[diFor1] THEN	
			IF __QUERYINTERFACE(AY_GROUPS[diFor1][LOWER_BOUND(AY_GROUPS[diFor1],1)],TEMP_ITF_CIRCUIT) THEN
				IF TEMP_ITF_CIRCUIT.GET_ANZ_RELEASE >= _uiHighestWorkloadCircuit THEN
					IF TEMP_ITF_CIRCUIT.GET_ANZ_RELEASE > _uiHighestWorkloadCircuit THEN
						_uiHighestWorkloadCircuit := TEMP_ITF_CIRCUIT.GET_ANZ_RELEASE; 
						(* Set Max Run Time To Min *)
						_udiMaxRunTimeTillOn := 16#0000;				
					END_IF;
					(* iterate Engine and Check if Avaiable and get the Minits *)
					FOR diFor2 := TEMP_ITF_CIRCUIT.UPPERBOUND TO TEMP_ITF_CIRCUIT.LOWERBOUND BY -1 DO
						TEMP_ITF_CIRCUIT.GET_ENGINE_STATE(	usiNr 			:= TO_USINT(diFor2),
															xAvaiable 		=> _xAvaiable,
															xRelease		=> _xRelease,
															rRelease		=> _rRelease,
															xAcknowledge 	=> _xAcknowledge,
															rAcknowledge 	=> _rAcknowledge,
															xLockDown 		=> _xLockDown,
															udiRunTime 		=> _udiRunTime,
															udiRunTimeTillOn=> _udiRunTimeTillOn);
						(* Get time if Running *)
						IF _xRelease THEN
							IF _udiRunTimeTillOn >= _udiMaxRunTimeTillOn THEN
								_udiMaxRunTimeTillOn 	:= _udiRunTimeTillOn;
								_diNextCircuitToOff 	:= diFor1;
								_diEngineHighestRunTime := diFor2;
							END_IF;			
						END_IF;						
					END_FOR;
				END_IF;
			END_IF;
		END_IF;
	END_FOR;
END_IF;
diNextCircuitToOffOut 	:= _diNextCircuitToOff;
diNextEngineToOffOut	:= _diEngineHighestRunTime;
END_METHOD

ACTION MANAGEMENT:
(* Wait til no Trig On *)
IF NOT xTrigOn THEN
	(* Get Next To Run *)
	GET_NEXT_ENGINE_TO_RUN(enTYPE_OF_ENGINE_MANAGEMENT := scParameter.fbiTypeOfEngineManagement.proValue, diNextCircuitToRunOut => diNextCircuitToRun, diNextEngineToRunOut => diNextEngineToRun);
END_IF;
(* Wait til no Trig Off *)
IF NOT xTrigOff THEN
	(* Get Next To Off *)
	GET_NEXT_ENGINE_TO_OFF(enTYPE_OF_ENGINE_MANAGEMENT := scParameter.fbiTypeOfEngineManagement.proValue, diNextCircuitToOffOut => diNextCircuitToOff, diNextEngineToOffOut => diNextEngineToOff);
END_IF;
(* Check if Engine Avaiable And Trig On *)
IF diNextCircuitToRun > 0 AND diNextEngineToRun > 0 THEN
	(* Check if Release *)
	IF xRelease AND iRelease > 0 AND NOT xReleaseStopp THEN
		(* Reaction on Group LockDown *)
		IF uiCountGroupLockDown > uiCountGroupLockDownOld AND NOT xLockDown THEN
			xTrigOn := TRUE;
			TP_ReleaseLock(IN	:= FALSE);
		(* Reaction on Engine LockDown *)
		ELSIF uiCountEngineLockDown > uiCountEngineLockDownOld AND NOT xLockDown THEN
			xTrigOn := TRUE;	
			TP_ReleaseLock(IN	:= FALSE);
		(* Reaction on Engine Off *)
		ELSIF uiCountEngineAcknowledge < uiCountEngineAcknowledgeOld AND iRelease = TO_INT(uiCountEngineAcknowledgeOld) AND NOT xLockDown THEN
			xTrigOn := TRUE;	
			TP_ReleaseLock(IN	:= FALSE);		
		(* Normal Trig Add Engine *)	
		ELSIF iRelease > iAcknowledge AND NOT TP_ReleaseLock.Q AND NOT xTrigOn THEN	
			// Resett Pulse before Trig
			TP_ReleaseLock(IN	:= FALSE);
			xTrigOn 			:= TRUE;
		END_IF;
	ELSE
		xTrigOn := FALSE;
	END_IF;
END_IF;

(* Normal Release Lock *)
IF NOT xResettReleaseLock_VIS  AND xRelease THEN
	IF scParameter.fbtZuschaltSperrzeit.proValue > T#60S THEN
		TP_ReleaseLock(PT :=  scParameter.fbtZuschaltSperrzeit.proValue);
	ELSE
		TP_ReleaseLock(PT := T#60S);
	END_IF
ELSE
	TP_ReleaseLock(IN := FALSE,
				   PT := T#0MS);
	xResettReleaseLock_VIS	:= FALSE;
END_IF;
(* Check if Engine Avaiable and Trig Off *)
IF diNextCircuitToOff > 0 AND diNextEngineToOff > 0 THEN
	(* Check if Release *)
	IF xRelease THEN
		(* Resett *)
		IF iRelease = iAcknowledge THEN
			iTrigOffMax   := 0;
			iTrigOffCount := 0;	
			(* Prevent endless runing of Engine if Relese is reduced to early and circuit is not already running *)
			IF xTrigOn THEN
				xTrigOn := FALSE;
				xTrigOff := TRUE;
				diNextCircuitToOff := diNextCircuitToRun;
				diNextEngineToOff  := diNextEngineToRun;			
			END_IF
		(* Normal Reduction *)
		ELSIF iRelease < iAcknowledge THEN
			// Reduce if redduce request during normal state or during start of engine
			IF  iRelease < iReleaseOld OR iAcknowledge > iAcknowledgeOld THEN	
				iTrigOffMax := MIN(iAcknowledge,iTrigOffMax + iReleaseOld - iRelease);
			END_IF
			IF iTrigOffCount < iTrigOffMax THEN
				iTrigOffCount := iTrigOffCount + 1;
				xTrigOff := TRUE;
			END_IF;
		END_IF;
	ELSE
		xTrigOff := FALSE;
	END_IF;
END_IF;

(* Set Release Array *)
FOR diFor1 := LOWER_BOUND(AY_GROUPS,1) TO UPPER_BOUND(AY_GROUPS,1) DO 
	IF __QUERYINTERFACE(AY_GROUPS[diFor1][LOWER_BOUND(AY_GROUPS[diFor1],1)],TEMP_ITF_CIRCUIT) THEN
		IF NOT AY_GROUPS_xLOCKDOWN[diFor1] THEN
			IF TEMP_ITF_CIRCUIT.IS_RELEVANT_TO_RELEASE THEN
				(* Off if this Ciruit or Engine is the next Off *)
				IF xRelease AND diFor1 = diNextCircuitToOff AND xTrigOff THEN
					(* Stopp Engine*)
					TEMP_ITF_CIRCUIT.RELEASE_ENGINE(TO_USINT(diNextEngineToOff),FALSE);
					xTrigOff := FALSE;
					xTrigOn  := FALSE;
				END_IF;				
				(* Release if this Ciruit is the next and Trig *)
				IF xRelease AND diFor1 = diNextCircuitToRun AND xTrigOn AND iRelease > 0 THEN
					(* Check if Avaiable *)
					IF AY_GROUPS_xAVAIABLE[diFor1] OR AY_GROUPS_xReleaseCircuit[diFor1] THEN
						AY_GROUPS_xRELEASE[diFor1] := TRUE;
					END_IF;
					IF AY_GROUPS_xReleaseCircuit[diFor1] THEN
						(* Release Engine*)
						TEMP_ITF_CIRCUIT.RELEASE_ENGINE(TO_USINT(diNextEngineToRun),TRUE);
						xTrigOn 			:= FALSE;
						TP_ReleaseLock(IN	:= TRUE);
					ELSE
						TEMP_ITF_CIRCUIT.ALL_OFF();
					END_IF;
				ELSIF NOT xRelease OR TEMP_ITF_CIRCUIT.GET_ANZ_RELEASE = 0 OR iRelease = 0 THEN
					TEMP_ITF_CIRCUIT.ALL_OFF();
					AY_GROUPS_xRELEASE[diFor1] := FALSE;
				END_IF;		
			ELSE
				AY_GROUPS_xRELEASE[diFor1] := xRelease;
			END_IF;
		ELSE
			TEMP_ITF_CIRCUIT.ALL_OFF();
			AY_GROUPS_xRELEASE[diFor1] := FALSE;
		END_IF;
	ELSE
		AY_GROUPS_xRELEASE[diFor1] := FALSE;
	END_IF;
END_FOR;

(* Set HZ Scale *)
FOR diFor1 := LOWER_BOUND(AY_GROUPS,1) TO UPPER_BOUND(AY_GROUPS,1) DO 
	IF __QUERYINTERFACE(AY_GROUPS[diFor1][LOWER_BOUND(AY_GROUPS[diFor1],1)],TEMP_ITF_CIRCUIT) THEN
		IF TEMP_ITF_CIRCUIT.IS_RELEVANT_TO_RELEASE THEN
			TEMP_ITF_CIRCUIT.SET_HZ_SCALE(scHzRelease);
		END_IF;
	END_IF;
END_FOR;
(* Set Cyclic Speed if no Acknowledge Change*)
IF iAcknowledge = iAcknowledgeOld THEN
	FOR diFor1 := LOWER_BOUND(AY_GROUPS,1) TO UPPER_BOUND(AY_GROUPS,1) DO 
		IF __QUERYINTERFACE(AY_GROUPS[diFor1][LOWER_BOUND(AY_GROUPS[diFor1],1)],TEMP_ITF_CIRCUIT) THEN
			IF TEMP_ITF_CIRCUIT.IS_RELEVANT_TO_RELEASE THEN
				FOR diFor2 := TEMP_ITF_CIRCUIT.LOWERBOUND TO TEMP_ITF_CIRCUIT.UPPERBOUND DO
					TEMP_ITF_CIRCUIT.prorRelease := rRelease;
				END_FOR
			END_IF;
		END_IF;
	END_FOR;
END_IF;
END_ACTION

ACTION CHECK_RELEASE_CHANGE:
(* Not Avaiable if Changed *)
IF enCheck <> enCheckOld THEN
	xAvaiable := FALSE;
END_IF;
END_ACTION

ACTION UPDATE_AT_THE_END:
(* Set Status Release and Check *)
FOR diFor1 := LOWER_BOUND(AY_GROUPS,1) TO UPPER_BOUND(AY_GROUPS,1) DO
	FOR diFor2 := LOWER_BOUND(AY_GROUPS[diFor1],1) TO UPPER_BOUND(AY_GROUPS[diFor1],1) DO
		IF AY_GROUPS[diFor1][diFor2] <> 0 THEN
			AY_GROUPS[diFor1][diFor2].SET_OPERATION_MODES(enCheckIn := enCheck,enReleaseIn := enRelease);
		END_IF;
	END_FOR;	
END_FOR;
iAcknowledgeOld := iAcknowledge;
enReleaseOld 	:= enRelease;
enCheckOld	 	:= enCheck;
iReleaseOld		:= iRelease;
END_ACTION

ACTION ACKNOWLEDGE:
(* Resett *)
FOR diFor1 := LOWER_BOUND(AY_GROUPS,1) TO UPPER_BOUND(AY_GROUPS,1) DO
	AY_GROUPS_xACKNOWLEDG[diFor1] := TRUE;	
END_FOR;
(* Get Status Acknowledge *)
FOR diFor1 := LOWER_BOUND(AY_GROUPS,1) TO UPPER_BOUND(AY_GROUPS,1) DO
	diTempMemberCount := 0;
	FOR diFor2 := LOWER_BOUND(AY_GROUPS[diFor1],1) TO UPPER_BOUND(AY_GROUPS[diFor1],1) DO
		IF AY_GROUPS[diFor1][diFor2] <> 0 THEN
			diTempMemberCount := diTempMemberCount + 1;
			IF NOT AY_GROUPS[diFor1][diFor2].IS_NOT_RELEVANT_TO_RELEASE AND NOT AY_GROUPS[diFor1][diFor2].IS_NOT_RELEVANT_TO_ACKNOWLEDGE THEN
				IF NOT AY_GROUPS[diFor1][diFor2].proxACKNOWLEDGE THEN
					AY_GROUPS_xACKNOWLEDG[diFor1] := FALSE;	
				END_IF;
			END_IF;
		END_IF;
	END_FOR;	
	(* Not Acknowledge if only Group Leader Added to Group *)
	IF diTempMemberCount <= 1 THEN
		AY_GROUPS_xACKNOWLEDG[diFor1] := FALSE;	
	END_IF;
	IF __QUERYINTERFACE(AY_GROUPS[diFor1][LOWER_BOUND(AY_GROUPS[diFor1],1)],TEMP_ITF_CIRCUIT) THEN
		AY_GROUPS_iACKNOWLEDG[diFor1] := TO_INT(TEMP_ITF_CIRCUIT.GET_ANZ_ACKNOWLEDGE);
	ELSE
		AY_GROUPS_iACKNOWLEDG[diFor1] := 0;
	END_IF;
END_FOR;

(* Set Status Acknowledge of Manager*)
xAcknowledge := FALSE;
FOR diFor1 := LOWER_BOUND(AY_GROUPS,1) TO UPPER_BOUND(AY_GROUPS,1) DO
	IF AY_GROUPS_xACKNOWLEDG[diFor1] THEN
		xAcknowledge := TRUE;
	END_IF;
END_FOR;
iAcknowledge := 0;
uiCountEngineAcknowledgeOld := uiCountEngineAcknowledge;
FOR diFor1 := LOWER_BOUND(AY_GROUPS,1) TO UPPER_BOUND(AY_GROUPS,1) DO
	iAcknowledge := iAcknowledge + AY_GROUPS_iACKNOWLEDG[diFor1];
END_FOR;
uiCountEngineAcknowledge := TO_UINT(iAcknowledge);
rAcknowledge := 0;
FOR diFor1 := LOWER_BOUND(AY_GROUPS,1) TO UPPER_BOUND(AY_GROUPS,1) DO
	rAcknowledge := rAcknowledge + AY_GROUPS_rACKNOWLEDG[diFor1];
END_FOR;
END_ACTION

ACTION RELEASE:
(* Set Release in Time Prio*)
T_Temp_Max_CT := T#0MS;
FOR diFor1 := LOWER_BOUND(AY_GROUPS,1) TO UPPER_BOUND(AY_GROUPS,1) DO
	IF AY_GROUPS_xRELEASE[diFor1] AND NOT AY_GROUPS_xLOCKDOWN[diFor1] THEN
		(* Set Ready as Resett *)
		AY_GROUPS_xReleaseCircuit[diFor1] := TRUE;
		(* Get Longest Time Till Run *)
		FOR diFor2 := LOWER_BOUND(AY_GROUPS[diFor1],1)+ 1 TO UPPER_BOUND(AY_GROUPS[diFor1],1) DO
			IF AY_GROUPS[diFor1][diFor2] <> 0 THEN
				IF NOT AY_GROUPS[diFor1][diFor2].IS_NOT_RELEVANT_TO_RELEASE AND NOT AY_GROUPS[diFor1][diFor2].IS_NOT_RELEVANT_TO_ACKNOWLEDGE THEN
					IF NOT AY_GROUPS[diFor1][diFor2].proxACKNOWLEDGE THEN
						IF __QUERYINTERFACE(AY_GROUPS[diFor1][diFor2],TEMP_ITF_HYDRA) THEN
							(* Get Longest Time till Run *)
							IF TEMP_ITF_HYDRA.CALCULATET_TIME_TILL_RUN >= T_Temp_Max_CT THEN
								T_Temp_Max_CT := TEMP_ITF_HYDRA.CALCULATET_TIME_TILL_RUN;
								AY_GROUPS_AyPosMaxCT[diFor1] := diFor2;
							END_IF
						END_IF;
						(* Set Not Ready To Release *)
						AY_GROUPS_xReleaseCircuit[diFor1] := FALSE;
					END_IF;
				END_IF;
			END_IF;
		END_FOR;	
		
		(* Relese Longest CT *)
		IF __QUERYINTERFACE(AY_GROUPS[diFor1][AY_GROUPS_AyPosMaxCT[diFor1]],TEMP_ITF_HYDRA_MAX_CT) THEN
			TEMP_ITF_HYDRA_MAX_CT.metSetRelease(TO_USINT(diFor1),TRUE);
		END_IF;
		  
		(* Release in Order of Max CT *)
		FOR diFor2 := LOWER_BOUND(AY_GROUPS[diFor1],1)+ 1 TO UPPER_BOUND(AY_GROUPS[diFor1],1) DO
			IF AY_GROUPS[diFor1][diFor2] <> 0 THEN
				(* check if relevant *)
				IF NOT AY_GROUPS[diFor1][diFor2].IS_NOT_RELEVANT_TO_RELEASE THEN
					IF __QUERYINTERFACE(AY_GROUPS[diFor1][diFor2],TEMP_ITF_HYDRA) THEN
						IF NOT AY_GROUPS[diFor1][diFor2].IS_NOT_RELEVANT_TO_ACKNOWLEDGE THEN	 
							IF NOT AY_GROUPS[diFor1][diFor2].proxACKNOWLEDGE THEN
							   IF __QUERYINTERFACE(AY_GROUPS[diFor1][AY_GROUPS_AyPosMaxCT[diFor1]],TEMP_ITF_HYDRA_MAX_CT) THEN
									(* Relese If Calculatet Time is Lower Estimatet Max *)
									IF TEMP_ITF_HYDRA.CALCULATET_TIME_TILL_RUN >= TEMP_ITF_HYDRA_MAX_CT.ESTIMATET_TIME_TILL_RUN THEN
										TEMP_ITF_HYDRA.metSetRelease(TO_USINT(diFor1),TRUE);
									END_IF;		
								ELSE
									TEMP_ITF_HYDRA.metSetRelease(TO_USINT(diFor1),TRUE);
								END_IF;
							ELSE
								TEMP_ITF_HYDRA.metSetRelease(TO_USINT(diFor1),TRUE);
							END_IF;
						ELSE
							TEMP_ITF_HYDRA.metSetRelease(TO_USINT(diFor1),TRUE);
						END_IF
					END_IF;
				ELSE
					IF __QUERYINTERFACE(AY_GROUPS[diFor1][diFor2],TEMP_ITF_HYDRA) THEN
						(* If not Relevant Off *)
						TEMP_ITF_HYDRA.metSetRelease(TO_USINT(diFor1),FALSE);
					END_IF;
				END_IF;
			END_IF;
		END_FOR;	
		(* Release Leader *)
		IF AY_GROUPS[diFor1][LOWER_BOUND(AY_GROUPS[diFor1],1)]	<> 0 THEN
			IF __QUERYINTERFACE(AY_GROUPS[diFor1][LOWER_BOUND(AY_GROUPS[diFor1],1)],TEMP_ITF_CIRCUIT) THEN
				IF TEMP_ITF_CIRCUIT.IS_RELEVANT_TO_RELEASE THEN
					IF AY_GROUPS_xReleaseCircuit[diFor1] THEN
						TEMP_ITF_CIRCUIT.metSetRelease(TRUE);
					ELSE
						(* If not Ready to Release Off*)
						TEMP_ITF_CIRCUIT.metSetRelease(FALSE);
					END_IF
				ELSE
					(* If not Relevant Off *)
					TEMP_ITF_CIRCUIT.metSetRelease(FALSE);
				END_IF;	
			END_IF;
		END_IF;
	ELSE
		(* All Off *)
		FOR diFor2 := LOWER_BOUND(AY_GROUPS[diFor1],1) TO UPPER_BOUND(AY_GROUPS[diFor1],1) DO
			IF __QUERYINTERFACE(AY_GROUPS[diFor1][diFor2],TEMP_ITF_CIRCUIT) THEN
				TEMP_ITF_CIRCUIT.metSetRelease(FALSE);
				
			ELSIF __QUERYINTERFACE(AY_GROUPS[diFor1][diFor2],TEMP_ITF_HYDRA) THEN
				TEMP_ITF_HYDRA.metSetRelease(TO_USINT(diFor1),FALSE);
			END_IF;
		END_FOR;	
		(* Set Not Ready To Release *)
		AY_GROUPS_xReleaseCircuit[diFor1] := FALSE;		
	END_IF
END_FOR;
END_ACTION

ACTION LOCKDOWN:
(* Resett *)
uiCountGroupLockDownOld := uiCountGroupLockDown;
uiCountGroupLockDown := 0;
FOR diFor1 := LOWER_BOUND(AY_GROUPS,1) TO UPPER_BOUND(AY_GROUPS,1) DO
	AY_GROUPS_xLOCKDOWN[diFor1] := FALSE;	
END_FOR;
(* Get Status LockDown *)
FOR diFor1 := LOWER_BOUND(AY_GROUPS,1) TO UPPER_BOUND(AY_GROUPS,1) DO
	FOR diFor2 := LOWER_BOUND(AY_GROUPS[diFor1],1) TO UPPER_BOUND(AY_GROUPS[diFor1],1) DO
		IF AY_GROUPS[diFor1][diFor2] <> 0 THEN
			IF NOT AY_GROUPS[diFor1][diFor2].IS_NOT_RELEVANT_TO_RELEASE THEN
				IF AY_GROUPS[diFor1][diFor2].proxLockDown THEN
					AY_GROUPS_xLOCKDOWN[diFor1] := TRUE;
					IF diNextCircuitToRun = diFor1 AND xTrigOn THEN
						xTrigOn := FALSE;
					END_IF;
				END_IF;
			END_IF;
		END_IF;
	END_FOR;	
END_FOR;

(* LockDown Group *)
xLockDown := FALSE;
FOR diFor1 := LOWER_BOUND(AY_GROUPS,1) TO UPPER_BOUND(AY_GROUPS,1) DO
	IF AY_GROUPS[diFor1][0] <> 0 THEN
		(* Lockdown wenn keine Gruppe *)
		IF AY_GROUPS_xLOCKDOWN[diFor1] THEN 
			xLockDown := TRUE;
			uiCountGroupLockDown := uiCountGroupLockDown + 1;
		END_IF;
	END_IF;
END_FOR
FOR diFor1 := LOWER_BOUND(AY_GROUPS,1) TO UPPER_BOUND(AY_GROUPS,1) DO
	IF AY_GROUPS[diFor1][0] <> 0 THEN
		(* Lockdown wenn keine Gruppe *)
		IF NOT AY_GROUPS_xLOCKDOWN[diFor1] AND (AY_GROUPS_xAVAIABLE[diFor1] OR AY_GROUPS_xACKNOWLEDG[diFor1]) THEN 
			xLockDown := FALSE;
		END_IF;
	END_IF;
END_FOR;

(* Get Status LockDown Engine*)
uiCountEngineLockDownOld := uiCountEngineLockDown;
uiCountEngineLockDown := 0;
FOR diFor1 := LOWER_BOUND(AY_GROUPS,1) TO UPPER_BOUND(AY_GROUPS,1) DO
	IF __QUERYINTERFACE(AY_GROUPS[diFor1][LOWER_BOUND(AY_GROUPS[diFor1],1)],TEMP_ITF_CIRCUIT) THEN
		uiCountEngineLockDown := uiCountEngineLockDown + TEMP_ITF_CIRCUIT.GET_ANZ_LOCKDOWN;
	END_IF;
END_FOR;
END_ACTION

ACTION AVAIABLE:
(* Resett *)
FOR diFor1 := LOWER_BOUND(AY_GROUPS,1) TO UPPER_BOUND(AY_GROUPS,1) DO
	AY_GROUPS_xAVAIABLE[diFor1] := TRUE;	
END_FOR;
(* Get Status Avaiable of Groups*)
FOR diFor1 := LOWER_BOUND(AY_GROUPS,1) TO UPPER_BOUND(AY_GROUPS,1) DO
	diTempMemberCount := 0;
	FOR diFor2 := LOWER_BOUND(AY_GROUPS[diFor1],1) TO UPPER_BOUND(AY_GROUPS[diFor1],1) DO
		IF AY_GROUPS[diFor1][diFor2] <> 0 THEN
			diTempMemberCount := diTempMemberCount + 1;
			IF NOT AY_GROUPS[diFor1][diFor2].IS_NOT_RELEVANT_TO_CHECK THEN
				IF NOT AY_GROUPS[diFor1][diFor2].proxAvaiable THEN
					AY_GROUPS_xAVAIABLE[diFor1] := FALSE;	
				END_IF;
			END_IF;
		END_IF;
	END_FOR;	
	(* Not Avaiable if only Group Leader Added to Group or Empty Group*)
	IF diTempMemberCount <= 1 THEN
		AY_GROUPS_xAVAIABLE[diFor1] := FALSE;	
	END_IF;
	IF __QUERYINTERFACE(AY_GROUPS[diFor1][LOWER_BOUND(AY_GROUPS[diFor1],1)],TEMP_ITF_CIRCUIT) THEN
		AY_GROUPS_iAVAIABLE[diFor1] := TO_INT(TEMP_ITF_CIRCUIT.GET_ANZ_AVAIABLE);
	ELSE
		AY_GROUPS_iAVAIABLE[diFor1] := 0;
	END_IF;	
END_FOR;
(* Set Status Avaiable of Manager*)
xAvaiable := FALSE;
FOR diFor1 := LOWER_BOUND(AY_GROUPS,1) TO UPPER_BOUND(AY_GROUPS,1) DO
	IF AY_GROUPS_xAVAIABLE[diFor1] THEN
		xAvaiable := TRUE;
	END_IF;
END_FOR;

iAvaiable := 0;
FOR diFor1 := LOWER_BOUND(AY_GROUPS,1) TO UPPER_BOUND(AY_GROUPS,1) DO
	iAvaiable := iAvaiable + AY_GROUPS_iAVAIABLE[diFor1];
END_FOR;
END_ACTION

METHOD ADD_CLIENT : BOOL
VAR_INPUT
	ITF_GROUP_BASE_IN	:	ITF_GROUPBASE;
END_VAR
VAR
	ITF_CIRCUIT_QUERRY	:	ITF_CIRCUIT;
	usiCircuitNr		:	USINT;
	ITF_HYDRA_QUERRY	:	ITF_HYDRA;
	xFailToAdd			:	BOOL;
	xExist				:	BOOL;
	xRegroup			:	BOOL;
	diForTemp1			:	DINT;
	diForTemp2			:	DINT;
	diForTemp3			:	DINT;
	diAddIn				:	DINT;
END_VAR
(* ADD CIRCUIT *)
IF __QUERYINTERFACE(ITF_GROUP_BASE_IN,ITF_CIRCUIT_QUERRY) THEN
	usiCircuitNr := ITF_CIRCUIT_QUERRY.CIRCUIT_NR;
	IF usiCircuitNr >= 1 AND usiCircuitNr <= GVL_CONSTANT.MAX_GROUPS THEN 
		IF AY_GROUPS[usiCircuitNr][0] = 0 THEN
			__QUERYINTERFACE(ITF_CIRCUIT_QUERRY,AY_GROUPS[usiCircuitNr][0]);
		ELSIF AY_GROUPS[usiCircuitNr][0] = ITF_GROUP_BASE_IN THEN
			ADD_CLIENT := TRUE;	
		ELSE
			ADD_CLIENT := FALSE;
		END_IF;
	END_IF;
(* ADD HYDRA *)
ELSIF __QUERYINTERFACE(ITF_GROUP_BASE_IN,ITF_HYDRA_QUERRY) THEN
	(* Check if is ADDED *)
	IF NOT ITF_HYDRA_QUERRY.IS_ADDED_TO_NESSESARY THEN
		FOR diForTemp1 := LOWER_BOUND(AY_GROUPS,1) TO UPPER_BOUND(AY_GROUPS,1) DO
			(* Reset Exist *)
			xExist := FALSE;
			(* Get Group Member *)
			IF ITF_HYDRA_QUERRY.MEMBER_OF(TO_USINT(diForTemp1)) THEN
				FOR diForTemp2 := LOWER_BOUND(AY_GROUPS[diForTemp1],1) TO UPPER_BOUND(AY_GROUPS[diForTemp1],1) DO
					IF AY_GROUPS[diForTemp1][diForTemp2] = ITF_GROUP_BASE_IN THEN
						xExist  := TRUE;
					END_IF;
				END_FOR;
				(* Add if not Exist *)
				IF NOT xExist THEN 
					IF aydiSyncG[diForTemp1] <> 0 THEN
						diAddIn  := __XADD(ADR(aydiSyncG[diForTemp1]),1);
						IF diAddIn >= 1 AND diAddIn <= UPPER_BOUND(AY_GROUPS[diForTemp1],1) THEN
							__QUERYINTERFACE(ITF_HYDRA_QUERRY,AY_GROUPS[diForTemp1][diAddIn]);
						ELSE
							xFailToAdd := TRUE;	
							ADD_CLIENT := FALSE;
						END_IF
					ELSE	
						xFailToAdd := TRUE;
						ADD_CLIENT := FALSE;
					END_IF;
				END_IF;
			ELSE
				FOR diForTemp2 := LOWER_BOUND(AY_GROUPS[diForTemp1],1) TO UPPER_BOUND(AY_GROUPS[diForTemp1],1) DO
					IF AY_GROUPS[diForTemp1][diForTemp2] = ITF_GROUP_BASE_IN THEN
						AY_GROUPS[diForTemp1][diForTemp2] := 0;
						FOR diForTemp3 := diForTemp2 TO UPPER_BOUND(AY_GROUPS[diForTemp1],1)-1 DO 
							AY_GROUPS[diForTemp1][diForTemp3] := AY_GROUPS[diForTemp1][diForTemp3+1];	
						END_FOR
						diAddIn  := __XADD(ADR(aydiSyncG[diForTemp1]),-1);
					END_IF;
				END_FOR;				
			END_IF
		END_FOR;
		ITF_HYDRA_QUERRY.IS_ADDED_TO_NESSESARY := NOT xFailToAdd;
	END_IF;	
ELSE
	ADD_CLIENT := FALSE;
END_IF;
END_METHOD

ACTION actParameter:
fbConfigFile();

scParameter.fbiTypeOfEngineManagement	(_usiParaNr := 1,	_WertInit := 0,		_MinInit := 0,	_MaxInit := 2,	itfConfigFb := fbConfigFile);
scParameter.fbtZuschaltSperrzeit		(_usiParaNr := 2,	_WertInit := T#5M,	_MinInit :=  ,	_MaxInit :=	 ,	itfConfigFb := fbConfigFile);
END_ACTION

END_FUNCTION_BLOCK

// 40 Visualizations/Dialog/DIA_MANAGER
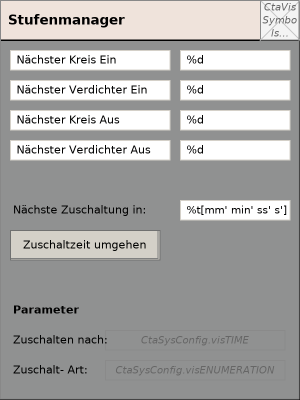
VISUALIZATION DIA_MANAGER  // 300x400
VAR_IN_OUT
	{attribute 'VAR_IN_OUT_AS_POINTER'}
	MANAGER_DIA			:	MANAGER;
END_VAR
    Rectangle (0,0 300x40)
    Rectangle (0,40 300x360)
    Button (10,230 150x30), "Zuschaltzeit umgehen"
        toggle MANAGER_DIA.xResettReleaseLock_VIS
    Textfield (10,50 160x20), "Nächster Kreis Ein"
    Textfield (10,80 160x20), "Nächster Verdichter Ein"
    Textfield (10,140 160x20), "Nächster Verdichter Aus"
    Textfield (10,110 160x20), "Nächster Kreis Aus"
    Textfield (180,50 110x20), "%d", text variable: MANAGER_DIA.diNextCircuitToRun
    Textfield (180,80 110x20), "%d", text variable: MANAGER_DIA.diNextEngineToRun
    Textfield (180,110 110x20), "%d", text variable: MANAGER_DIA.diNextCircuitToOff
    Textfield (180,140 110x20), "%d", text variable: MANAGER_DIA.diNextEngineToOff
    Frame (105,330 180x20)
        shows CtaSysConfig.visTIME(visfbTIMEIn := MANAGER_DIA.scParameter.fbtZuschaltSperrzeit)
    Frame (105,360 180x20), text list: 'TypeOfEngineManagement', text index: CtaSysConfig.fcGetEnumerationId(MANAGER_DIA.scParameter.fbiTypeOfEngineManagement)
        shows CtaSysConfig.visENUMERATION(visfbENUIn := MANAGER_DIA.scParameter.fbiTypeOfEngineManagement)
    Label (10,330 150x20), "Zuschalten nach:"
    Label (10,360 150x20), "Zuschalt- Art:"
    Textfield (180,200 110x20), "%t[mm' min' ss' s']", text variable: (MANAGER_DIA.scParameter.fbtZuschaltSperrzeit.proValue - MANAGER_DIA.TP_ReleaseLock.ET)
    Textfield (10,200 160x20), "Nächste Zuschaltung in:"
    Textfield (10,300 160x20), "Parameter"
    Image (260,0 40x40), image: CtaVisSymbols.ImagePool.close_solo_black
        OnMouseClick:  Dialog=Current Dialog, Result=OK, NumpadKeypadSet=True
    Label (5,10 150x20), "Stufenmanager"
END_VISUALIZATION

// 40 Visualizations/VIS_Manager_rEck
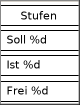
VISUALIZATION VIS_Manager_rEck  // 80x105
VAR_IN_OUT
	MANAGER_IN		:	MANAGER;
END_VAR
    Textfield (0,1 80x105)
    Textfield (0,6 78x20), "Stufen"
    Textfield (0,30 78x20), "Soll %d", text variable: MANAGER_IN.iRelease
    Textfield (0,55 78x20), "Ist %d", text variable: MANAGER_IN.iAcknowledge
    Textfield (0,81 78x20), "Frei %d", text variable: MANAGER_IN.iAvaiable
    Rectangle (0,0 80x105)
        OnMouseClick:  Dialog=DIA_MANAGER, Parameters={MANAGER_DIA: MANAGER_IN}, Selected={0: }, OpenCentered=True
    Line (0,30) (79,30)
    Line (0,50) (79,50)
    Line (0,55) (79,55)
    Line (0,75) (79,75)
    Line (0,81) (79,81)
    Line (0,101) (79,101)
    Line (0,5) (79,5)
    Line (0,25) (79,25)
END_VISUALIZATION

// 40 Visualizations/VIS_Manager
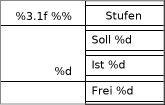
VISUALIZATION VIS_Manager  // 165x105
VAR_IN_OUT
	MANAGER_IN		:	MANAGER;
END_VAR
    Line (0,25) (157,25)
    Line (0,81) (158,81)
    Rectangle (15,65 60x13), "%d", text variable: MANAGER_IN.iRelease
    Frame (85,0 80x105)
        shows VIS_Manager_rEck(MANAGER_IN := MANAGER_IN)
    Rectangle (15,10 60x13), "%3.1f %%", text variable: MANAGER_IN.rRelease
END_VISUALIZATION

(* text list TypeOfEngineManagement (id | default)
  0 | RUN 1BY1
  1 | RUN EQUAL
   |  *)
